{attribute 'qualified_only'}
{attribute 'strict'}
TYPE E_EpicsHomeCmd :
    // Defines the valid options for homing in FB_MotionStage
(
    LOW_LIMIT := 1, // Low limit switch
    HIGH_LIMIT := 2, // High limit switch
    HOME_VIA_LOW := 3, // Home switch via low switch
    HOME_VIA_HIGH := 4, // Home switch via high switch
    ABSOLUTE_SET := 15, // Set here to be fHomePosition
    // MCS2
    AutoMethod := -1, // DS402 Auto method; referencing routine set by positioner type
    CURRENT_POSITION_METHOD := 37,
    NONE := -99 // Do not home, ever
) := NONE;
END_TYPE

(* stored: Version 1.1.0.1
   DUT E_EpicsHomeCmd: Id {5b99003f-e7b7-4d14-9ac5-0be5ae1ff947} *)
